FUNCTION_BLOCK OPC_UA_READ (* Read value from OPC UA server *)
  (* Standard: OPC UA; Function: Reader *)
  (* Version 1.0, 2015-11-08, Slavomir Kozar, Certicon *)
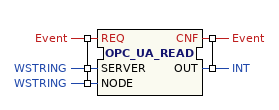
  EVENT_INPUT
    REQ WITH SERVER, NODE; (* Normal Execution Request *)
  END_EVENT
  EVENT_OUTPUT
    CNF WITH OUT; (* Execution Confirmation *)
  END_EVENT
  VAR_INPUT
    SERVER : WSTRING; (* OPC UA server address:port *)
    NODE : WSTRING; (* UPC UA Node ID *)
  END_VAR
  VAR_OUTPUT
    OUT : INT; (* Readed data *)
  END_VAR
END_FUNCTION_BLOCK
